# EPICS substitutions: db/Beckhoff_9XXX/ecmcEL9227-5500.substitutions
file "ecmcEL9227-5500-chX.template"
{
    pattern {CH_ID}
            {01   }
            {02   }
}
